{attribute addProperty BoxType ""}
{attribute addProperty Id "_defaultSyncUnitTasks_97D7B59B216270A_0022_EP9224_0037_0017SyncUnitTasks_97D7B59B216270"}
{attribute addProperty CRC "2845800459"}
{attribute addProperty SizeInBites "432"}
{attribute addProperty SizeInBytes "54"}
TYPE SyncUnits_A99F780B :
STRUCT
	{attribute addProperty Name "_default"}
	_default : SyncUnitTasks_97D7B59B;
	{attribute addProperty Name "A_0022_EP9224_0037_0017"}
	A_0022_EP9224_0037_0017 : SyncUnitTasks_97D7B59B;
END_STRUCT
END_TYPE

(* stored: Version 1.2.0.0, ProductVersion 3.1.4024.9
   DUT SyncUnits_A99F780B: Id {b1e5eadf-b13e-4a94-a8d6-83dea403d48f} *)
